FUNCTION_BLOCK E_DELAY_V_D (* Composite Function Block Type *)
  (* Standard: 61499-2 *)
  (* Version 0.0, 2/4/2026, SESA713705, Schneider Electric, template *)
  PACKAGE SE.Nereda;
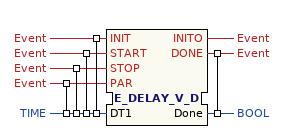
  EVENT_INPUT
    INIT WITH DT1;
    START WITH DT1; (* Begin Delay *)
    STOP WITH DT1; (* Cancel Delay *)
    PAR WITH DT1;
  END_EVENT
  EVENT_OUTPUT
    INITO;
    DONE WITH Done; (* Input changed *)
  END_EVENT
  VAR_INPUT
    DT1 : TIME; (* Delay Time *)
  END_VAR
  VAR_OUTPUT
    Done : BOOL; (* Output value *)
  END_VAR
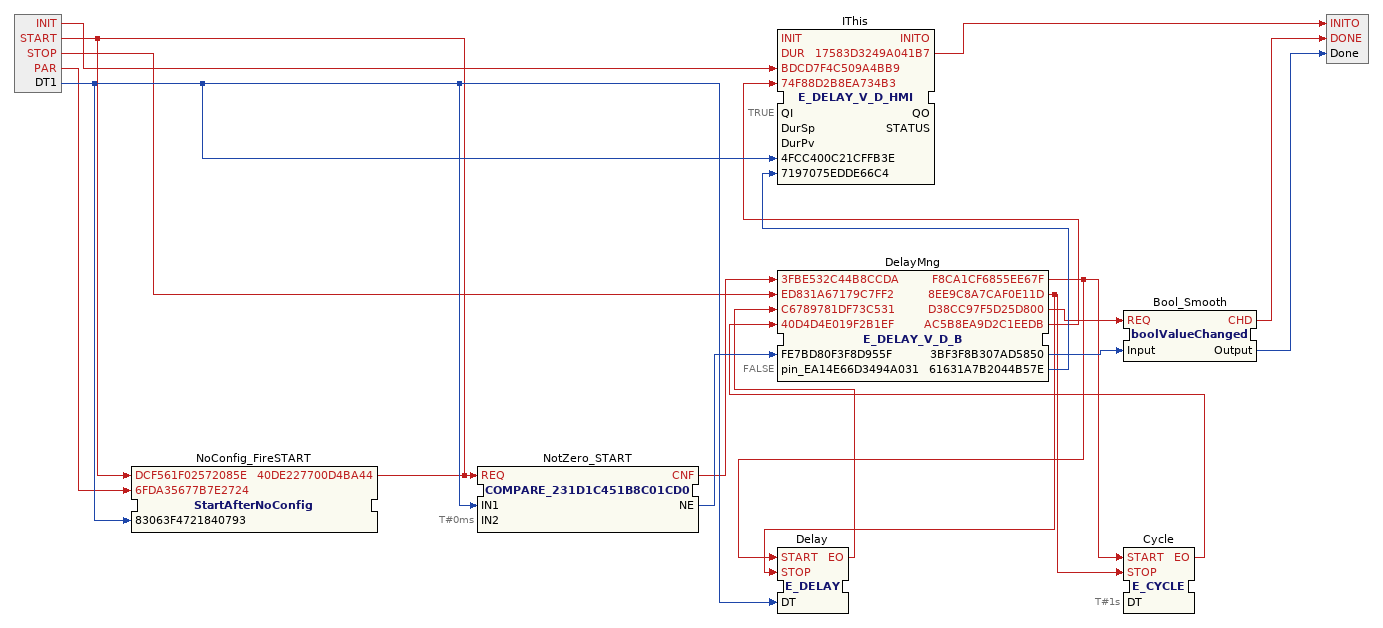
  FBS
    Bool_Smooth : boolValueChanged;
    IThis : E_DELAY_V_D_HMI(QI := TRUE);
    DelayMng : E_DELAY_V_D_B(pin_EA14E66D3494A031 := FALSE);
    Delay : E_DELAY;
    Cycle : E_CYCLE(DT := T#1s);
    NotZero_START : COMPARE_231D1C451B8C01CD0(IN2 := T#0ms); {SET_ATTRIBUTE(Configuration.GenericFBType.InterfaceParams, Runtime.Standard#CNT:=2;IN${CNT$}:TIME)}
    NoConfig_FireSTART : StartAfterNoConfig;
  END_FBS
  EVENT_CONNECTIONS
    Bool_Smooth.CHD TO DONE;
    INIT TO IThis.BDCD7F4C509A4BB9;
    IThis.17583D3249A041B7 TO INITO;
    START TO NoConfig_FireSTART.DCF561F02572085E;
    DelayMng.F8CA1CF6855EE67F TO Delay.START;
    DelayMng.F8CA1CF6855EE67F TO Cycle.START;
    DelayMng.8EE9C8A7CAF0E11D TO Delay.STOP;
    DelayMng.8EE9C8A7CAF0E11D TO Cycle.STOP;
    DelayMng.D38CC97F5D25D800 TO Bool_Smooth.REQ;
    DelayMng.AC5B8EA9D2C1EEDB TO IThis.74F88D2B8EA734B3;
    NotZero_START.CNF TO DelayMng.3FBE532C44B8CCDA;
    STOP TO DelayMng.ED831A67179C7FF2;
    Delay.EO TO DelayMng.C6789781DF73C531;
    Cycle.EO TO DelayMng.40D4D4E019F2B1EF;
    START TO NotZero_START.REQ;
    NoConfig_FireSTART.40DE227700D4BA44 TO NotZero_START.REQ;
    PAR TO NoConfig_FireSTART.6FDA35677B7E2724;
  END_CONNECTIONS
  DATA_CONNECTIONS
    Bool_Smooth.Output TO Done;
    DT1 TO IThis.4FCC400C21CFFB3E;
    DT1 TO Delay.DT;
    DT1 TO NotZero_START.IN1;
    DelayMng.3BF3F8B307AD5850 TO Bool_Smooth.Input;
    DelayMng.61631A7B2044B57E TO IThis.7197075EDDE66C4;
    NotZero_START.NE TO DelayMng.FE7BD80F3F8D955F;
    DT1 TO NoConfig_FireSTART.83063F4721840793;
  END_CONNECTIONS
END_FUNCTION_BLOCK
